FUNCTION_BLOCK PAClassPhysicalBase EXTENDS PAClassAlarmingBase IMPLEMENTS IRouteableComponent
VAR_INPUT
END_VAR
VAR_OUTPUT
END_VAR
VAR	
	_OperatingMode : PAOperatingModeEnum;
	_ReqOperatingMode : PAOperatingModeEnum;
	_Points : ARRAY [1..GCL.cPointMAX] OF IACPoint;
END_VAR

METHOD PUBLIC AddPoint : BOOL
VAR_INPUT
	point : IACPoint;
END_VAR
VAR
	i: INT;
END_VAR
IF point = 0 THEN
	Addpoint := FALSE;
	RETURN;
END_IF
// 1. Check if point already exists in the array because of online change
FOR i:=1 TO GCL.cPointMAX BY 1
  DO
    IF _points[i] <> 0 THEN
		IF _points[i].ACUrl = point.ACUrl THEN
			AddPoint := FALSE;
			RETURN;			
		END_IF
	ELSE
		EXIT;
	END_IF
END_FOR;
// 2. If the point doesn't exist, add to _points-List
FOR i:=1 TO GCL.cPointMAX BY 1
  DO
    IF _points[i] = 0 THEN
		AddPoint := TRUE;
		_points[i] := point;
		EXIT;
	END_IF
END_FOR;
END_METHOD

METHOD PUBLIC FB_postinit
VAR_INPUT
		root : IACVariobatch;
END_VAR
VAR
	i: INT;
END_VAR
SUPER^.FB_postinit(root);
root.OnPropertyChangedInt(THIS^, 10, _OperatingMode);
root.OnPropertyChangedInt(THIS^, 11, _ReqOperatingMode);
FOR i:=1 TO GCL.cPointMAX BY 1
  DO
    IF _Points[i] <> 0 THEN
		_Points[i].FB_postinit(root);
	ELSE
		EXIT;
	END_IF
END_FOR;
END_METHOD

METHOD PUBLIC FindObjectInChilds : IACObject
VAR_INPUT
	instanceID	: UDINT;
END_VAR
VAR
	i: INT;
	foundObject : IACObject;
	prevPoint : IACPoint;
	currentPoint : IACPoint;
END_VAR
foundObject := 0;
prevPoint := 0;
currentPoint := 0;

FOR i:=1 TO GCL.cPointMAX BY 1
  DO
    IF _Points[i] <> 0 THEN
		currentPoint := _Points[i];
		IF currentPoint.InstanceID = instanceID THEN
			FindObjectInChilds := currentPoint;
			RETURN;
		ELSIF currentPoint.InstanceID > instanceID THEN
			IF prevPoint <> 0 THEN
				foundObject := prevPoint.FindObjectInChilds(instanceID);
				EXIT;
			ELSE
				foundObject := 0;
				EXIT;
			END_IF
		ELSE
			prevPoint := currentPoint;
		END_IF
	ELSE
		EXIT;
	END_IF
END_FOR;

IF foundObject <> 0 THEN
	FindObjectInChilds := foundObject;
	RETURN;
END_IF

foundObject := SUPER^.FindObjectInChilds(instanceID);
IF foundObject <> 0 THEN
	FindObjectInChilds := foundObject;
	RETURN;
END_IF

IF prevPoint <> 0 AND prevPoint.InstanceID < instanceID THEN
	FindObjectInChilds := prevPoint.FindObjectInChilds(instanceID);
	RETURN;
END_IF

FindObjectInChilds := 0;
END_METHOD

METHOD PUBLIC InvokeSetterEnum
VAR_INPUT
	PropertyID : INT;
	PropertyValue : INT;
END_VAR
SUPER^.InvokeSetterEnum(PropertyID, PropertyValue);
IF PropertyID = 10 THEN
	THIS^.OperatingMode := PropertyValue;
ELSIF PropertyID = 11 THEN	
	THIS^.ReqOperatingMode := PropertyValue;
END_IF
END_METHOD

METHOD PUBLIC IsEnabledSwitchToAutomatic : BOOL
VAR_INPUT
END_VAR
END_METHOD

METHOD PUBLIC IsEnabledSwitchToMaintenance : BOOL
VAR_INPUT
END_VAR
END_METHOD

METHOD PUBLIC IsEnabledSwitchToManual : BOOL
VAR_INPUT
END_VAR
END_METHOD

METHOD OnInitMemory
VAR_INPUT
		root : IACVariobatch;
END_VAR
RegisterProperty(root, 10, GCL.cSizeINT); // _OperatingMode
RegisterProperty(root, 11, GCL.cSizeINT); // _ReqOperatingMode
SUPER^.OnInitMemory(root);
END_METHOD

{attribute 'monitoring' := 'call'}
//{attribute 'TcRpcEnable'}
PROPERTY PUBLIC OperatingMode : PAOperatingModeEnum
GET
OperatingMode := _OperatingMode;
END_GET
SET
_OperatingMode := OperatingMode;
Root.OnPropertyChangedInt(THIS^, 10, _OperatingMode);
END_SET
END_PROPERTY

PROPERTY PUBLIC Points : ARRAY [1..GCL.cPointMAX] OF IACPoint
GET
Points := _Points;
END_GET
END_PROPERTY

{attribute 'monitoring' := 'call'}
//{attribute 'TcRpcEnable'}
PROPERTY PUBLIC ReqOperatingMode : PAOperatingModeEnum
GET
ReqOperatingMode := _ReqOperatingMode;
END_GET
SET
_ReqOperatingMode := ReqOperatingMode;
Root.OnPropertyChangedInt(THIS^, 11, _ReqOperatingMode);
OperatingMode := _ReqOperatingMode;
END_SET
END_PROPERTY

METHOD PUBLIC SwitchToAutomatic
VAR_INPUT
END_VAR
_OperatingMode := PAOperatingModeEnum.Automatic;
END_METHOD

METHOD PUBLIC SwitchToMaintenance
VAR_INPUT
END_VAR
_OperatingMode := PAOperatingModeEnum.Maintenance;
END_METHOD

METHOD PUBLIC SwitchToManual
VAR_INPUT
END_VAR
_OperatingMode := PAOperatingModeEnum.Manual;
END_METHOD

END_FUNCTION_BLOCK

(* stored: Version 1.1.0.1, ProductVersion 3.1.4024.6
   POU PAClassPhysicalBase: Id {0b90114a-dfa9-486f-a322-a512c18d6ff4}, SpecialFunc None
   Method AddPoint: Id {71ceecca-2103-4f98-9cb0-27735bf8acad}
   Method FB_postinit: Id {3191daa4-ee60-486c-9ccd-9f62810c8551}
   Method FindObjectInChilds: Id {0f40a72e-9cbf-44e3-a02d-69e4a42279d9}
   Method InvokeSetterEnum: Id {b8791738-5091-48fb-8dd4-7b282e84bdef}
   Method IsEnabledSwitchToAutomatic: Id {d24fafd1-0c8a-43b3-a3bd-bfebfd529819}
   Method IsEnabledSwitchToMaintenance: Id {b3ebff3a-bf00-439a-84da-7f470e9c2f37}
   Method IsEnabledSwitchToManual: Id {2362c883-2fca-44d6-8dcc-59caad907f40}
   Method OnInitMemory: Id {5c312e19-b34f-4cde-b412-1863f7b772ba}
   Property OperatingMode: Id {f1860551-a3b4-461f-b5d6-b4a01adbbc60}
   Get Get: Id {d2c2da21-6ee4-4a31-b03e-1ee9196d8f95}
   Set Set: Id {2c66f92e-620f-4048-9b0d-faa6cb0371af}
   Property Points: Id {81a6501a-4cc4-4196-9876-5f06ca44bbe5}
   Get Get: Id {255f661d-8bab-47c6-b1dd-100ded474bae}
   Property ReqOperatingMode: Id {c49f4ded-1e96-4972-904d-53bb183b601c}
   Get Get: Id {11e46c0b-4d69-45ee-9d52-8722aa9e6a89}
   Set Set: Id {6dc10bdd-5685-495b-a3d7-125f95dec2ed}
   Method SwitchToAutomatic: Id {3b64ded2-e2f1-4697-8ed0-a318a5286948}
   Method SwitchToMaintenance: Id {55968c0c-1abe-431b-b890-ba725f2f4417}
   Method SwitchToManual: Id {4c46cb75-5ccb-4759-ae89-fc5aaa8951c6} *)
